(* CODESYS project filling_station_1808.ecp

Project tree, tasks and I/O mapping:
  GenericDummyMasterDevice : Generic Master, WAGO, order no. None, version 1.0.0.0
  PFC200_CS_2ETH_RS : 750-8202 PFC200 2ETH RS, WAGO, order no. 0750-8202, version 1.4.1.22
    application Application
      libraries: ; Util, * (System); VisuDialogs, * (System)
      task PLC_Task (cyclic, interval t#10ms, priority 14) calls PLC_PRG
      task Visu_Task (cyclic, interval t#10ms, priority 14) calls VISU_PRG
      function CONVERT_PRESSURE_TO_LEVEL [ST]
      visualisation Visualization
      function READ_PRESSURE [ST]
      global variables GVL
      function XOR_MANUAL_AUTOMATIC_VALVE_CONTROL [ST]
      function READ_VALVE_POSITION [ST]
      function AVOID_SIMULT_VALVE_OPEN_AND_CLOSE [ST]
      program PLC_PRG [FBD]
      image pool ImagePool
      visualisation Visualization_1
      function ASSIGN_OUTPUTS [ST]
      visualisation Visualization_2
      function ACTUATOR [ST]
    DeviceAdapter
    Kbus : Kbus, WAGO, version 1.3.0.0
        unmapped channels: K-BUS diagnostics
      _8_DO_Generic : 075x-8DO, WAGO, order no. 075x-8DO, version 0.0.0.11
          settings: K-BUS Module slot index = 1
          output vbOpenSamsonValve : BOOL  // _OUT._OUT
          output vbCloseSamsonValve : BOOL  // _OUT._OUT
          output vbOpenDrainValveAbovePump : BOOL  // _OUT._OUT
          output vbSwitchOnPump : BOOL  // _OUT._OUT
          unmapped channels: _OUT
        DeviceAdapter
      _4_AI_0_10V_DC_s_e : 0750-0459, WAGO, order no. 0750-0459, version 0.0.0.11
          settings: K-BUS Module slot index = 2
          input  vwRawValvePosition : WORD  // _IW 1
          unmapped channels: _IW 2, _IW 3, _IW 4
        DeviceAdapter
      _2_AI_4_20mA_Diff_Measurement_Input : 0750-0492, WAGO, order no. 0750-0492, version 0.0.0.7
          settings: K-BUS Module slot index = 3
          input  vwRawPressure : WORD  // _IW 1
          unmapped channels: _IW 2
        DeviceAdapter
    MODBUS
      MODBUS : MODBUS, WAGO, order no. n/a, version 1.1.1.13
    Serial
      COM1 : COM1, WAGO, version 0.0.0.19
  e_DISPLAY_7300T_WP_10_1_1280x800_PIO1 : 0762-3003 e!DISPLAY 7300T - WP 10.1, WAGO, order no. 0762-3003, version 0.0.0.3
    DeviceAdapter
  libraries: WagoVisuIcons, 1.0.0.7 (WAGO)
  text list GlobalTextList
  5ce3da45-db07-42e7-a21c-a00fff4ed8f6|C:\Users\Alexander Wilms\Documents\Ausbildung\Hochschule Darmstadt\Master Electrical Engineering\1. Semester\Team Project\team-project\40_Implementation\hydraulics-schematic-simplified.png
  5ce3da45-db07-42e7-a21c-a00fff4ed8f6|C:\Users\Alexander Wilms\Documents\Ausbildung\Hochschule Darmstadt\Master Electrical Engineering\1. Semester\Team Project\team-project\30_Architecture\hydraulics-schematic-simplified.png
*)

// PFC200_CS_2ETH_RS/Application/GVL
VAR_GLOBAL
	vrWaterLevel:REAL;
	vrgrWaterLevel:ARRAY[1..16] OF REAL;
	vrStandardGravity:REAL:=9.81;
	viDensityWater:INT:=1000;
	vrValvePosition:REAL;
	vrValvePositionPercentage:REAL;
	vrValvePositionDesired:REAL;
	viPumpPowerPercentage:INT;
	vbManualValveControl:BOOL:=TRUE;
	vbAutomaticValveControl:BOOL:=FALSE;
	vbPreviousValveControl:STRING:='MANUAL';
	vbPreviousSamsonValveDirection:STRING:='STOP';
	vbStopSamsonValve:BOOL:=TRUE;
	vbOpenSamsonValveCtrl:BOOL;
	vbCloseSamsonValveCtrl:BOOL;
	vbOpenDrainValveBelowVessel:BOOL:=FALSE;
	vbOpenDrainValveAbovePumpCtrl:BOOL:=FALSE;
	vbSwitchOnPumpCtrl:BOOL:=FALSE;
	vbTrash: BOOL;
	vrController_Level_SP:REAL;
	vrController_PV:REAL;
	vbController_Manual_Mode:BOOL:=FALSE;
	vrController_Output:REAL;
	vrController_Output_reversed:REAL;
	Water_Valve_Open: BOOL;
	Water_Valve_Close: BOOL;
	PID_1: PID;
END_VAR

// PFC200_CS_2ETH_RS/Application/PLC_PRG
PROGRAM PLC_PRG
VAR
	PID_0: PID;
	TRASH: BOOL;
END_VAR

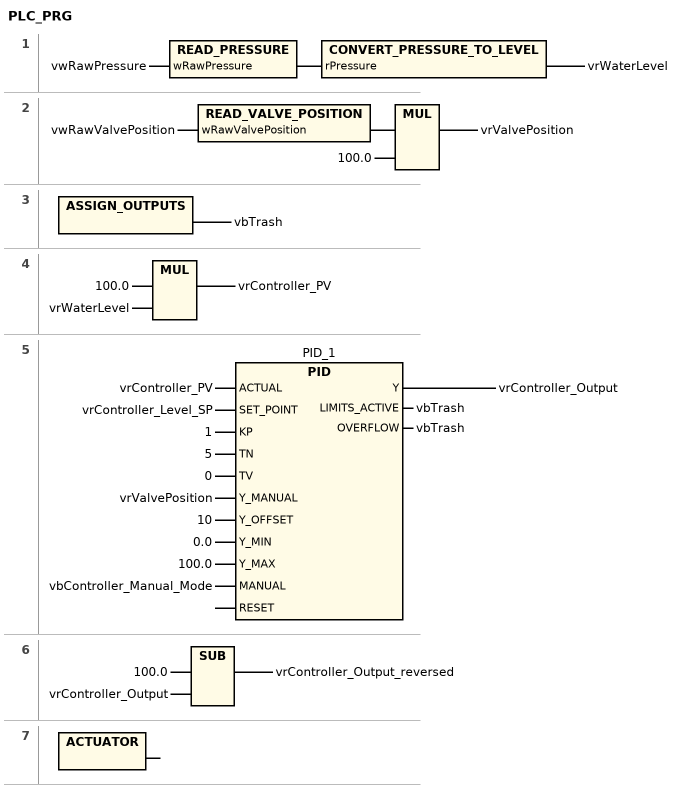
// NETWORK 1
vrWaterLevel := CONVERT_PRESSURE_TO_LEVEL(rPressure := READ_PRESSURE(wRawPressure := vwRawPressure));

// NETWORK 2
vrValvePosition := READ_VALVE_POSITION(wRawValvePosition := vwRawValvePosition) * 100.0;

// NETWORK 3
vbTrash := ASSIGN_OUTPUTS();

// NETWORK 4
vrController_PV := 100.0 * vrWaterLevel;

// NETWORK 5
PID_1(
    ACTUAL := vrController_PV,
    SET_POINT := vrController_Level_SP,
    KP := 1,
    TN := 5,
    TV := 0,
    Y_MANUAL := vrValvePosition,
    Y_OFFSET := 10,
    Y_MIN := 0.0,
    Y_MAX := 100.0,
    MANUAL := vbController_Manual_Mode,
    LIMITS_ACTIVE => vbTrash,
    OVERFLOW => vbTrash); // PID
vrController_Output := PID_1.Y;

// NETWORK 6
vrController_Output_reversed := 100.0 - vrController_Output;

// NETWORK 7
ACTUATOR();

END_PROGRAM

// PFC200_CS_2ETH_RS/Application/CONVERT_PRESSURE_TO_LEVEL
FUNCTION CONVERT_PRESSURE_TO_LEVEL : REAL
VAR_INPUT
	rPressure:REAL;
END_VAR
VAR
END_VAR

CONVERT_PRESSURE_TO_LEVEL := rPressure/viDensityWater/vrStandardGravity;

END_FUNCTION

// PFC200_CS_2ETH_RS/Application/READ_PRESSURE
FUNCTION READ_PRESSURE : REAL
VAR_INPUT
	wRawPressure:WORD;
END_VAR
VAR
END_VAR

READ_PRESSURE := WORD_TO_REAL((wRawPressure)*9800)/65535;

END_FUNCTION

// PFC200_CS_2ETH_RS/Application/READ_VALVE_POSITION
FUNCTION READ_VALVE_POSITION : REAL
VAR_INPUT
	wRawValvePosition:WORD;
END_VAR
VAR
END_VAR

READ_VALVE_POSITION := WORD_TO_REAL(wRawValvePosition)/65535;
vrValvePositionPercentage := READ_VALVE_POSITION*100;

END_FUNCTION

// PFC200_CS_2ETH_RS/Application/ASSIGN_OUTPUTS
FUNCTION ASSIGN_OUTPUTS : BOOL
VAR_INPUT
END_VAR
VAR
END_VAR

vbSwitchOnPump:=vbSwitchOnPumpCtrl;
vbOpenDrainValveAbovePump:=vbOpenDrainValveAbovePumpCtrl;
vbOpenSamsonValveCtrl:=vbOpenSamsonValve;
vbCloseSamsonValveCtrl:=vbCloseSamsonValve;
ASSIGN_OUTPUTS:=TRUE;

END_FUNCTION

// PFC200_CS_2ETH_RS/Application/ACTUATOR
FUNCTION ACTUATOR : BOOL
VAR_INPUT
END_VAR
VAR
END_VAR

IF (vrController_Output_reversed - vrValvePosition) <= 2 AND (  vrValvePosition - vrController_Output_reversed ) <=2
THEN
vbOpenSamsonValve:=vbOpenSamsonValve;
vbCloseSamsonValve:=vbCloseSamsonValve;
ELSIF
(vrController_Output_reversed - vrValvePosition) >2
THEN
vbOpenSamsonValve:=TRUE;
vbCloseSamsonValve:=FALSE;
ELSE
vbOpenSamsonValve:=FALSE;
vbCloseSamsonValve:=TRUE;
END_IF

END_FUNCTION

// PFC200_CS_2ETH_RS/Application/XOR_MANUAL_AUTOMATIC_VALVE_CONTROL
FUNCTION XOR_MANUAL_AUTOMATIC_VALVE_CONTROL : BOOL
VAR_INPUT
END_VAR
VAR
END_VAR

IF vbAutomaticValveControl AND vbManualValveControl THEN
	IF vbPreviousValveControl = 'MANUAL' THEN
			vbAutomaticValveControl := TRUE;
			vbManualValveControl := FALSE;
			vbPreviousValveControl := 'AUTOMATIC';
	ELSIF
			vbPreviousValveControl =  'AUTOMATIC' THEN
			vbAutomaticValveControl := FALSE;
			vbManualValveControl := TRUE;
			vbPreviousValveControl := 'MANUAL';
	END_IF
END_IF

XOR_MANUAL_AUTOMATIC_VALVE_CONTROL := TRUE;

END_FUNCTION

// PFC200_CS_2ETH_RS/Application/AVOID_SIMULT_VALVE_OPEN_AND_CLOSE
FUNCTION AVOID_SIMULT_VALVE_OPEN_AND_CLOSE : BOOL
VAR_INPUT
END_VAR
VAR
END_VAR

IF vbOpenSamsonValve AND vbStopSamsonValve THEN
	IF vbPreviousSamsonValveDirection = 'OPEN' THEN
		vbOpenSamsonValve := FALSE;
		vbStopSamsonValve := TRUE;
		vbCloseSamsonValve := FALSE;
		vbPreviousSamsonValveDirection := 'STOP';
	ELSIF vbPreviousSamsonValveDirection = 'STOP' THEN
		vbOpenSamsonValve := TRUE;
		vbStopSamsonValve := FALSE;
		vbCloseSamsonValve := FALSE;
		vbPreviousSamsonValveDirection := 'OPEN';
	END_IF
ELSIF vbStopSamsonValve AND vbCloseSamsonValve THEN
	IF vbPreviousSamsonValveDirection = 'STOP' THEN
		vbOpenSamsonValve := FALSE;
		vbStopSamsonValve := FALSE;
		vbCloseSamsonValve := TRUE;
		vbPreviousSamsonValveDirection := 'CLOSE';
	ELSIF vbPreviousSamsonValveDirection = 'CLOSE' THEN
		vbOpenSamsonValve := FALSE;
		vbStopSamsonValve := TRUE;
		vbCloseSamsonValve := FALSE;
		vbPreviousSamsonValveDirection := 'STOP';
	END_IF
ELSIF vbOpenSamsonValve AND vbCloseSamsonValve THEN
	IF vbPreviousSamsonValveDirection = 'OPEN' THEN
		vbOpenSamsonValve := FALSE;
		vbStopSamsonValve := FALSE;
		vbCloseSamsonValve := TRUE;
		vbPreviousSamsonValveDirection := 'CLOSE';
	ELSIF vbPreviousSamsonValveDirection = 'CLOSE' THEN
		vbOpenSamsonValve := TRUE;
		vbStopSamsonValve := FALSE;
		vbCloseSamsonValve := FALSE;
		vbPreviousSamsonValveDirection := 'OPEN';
	END_IF
END_IF

AVOID_SIMULT_VALVE_OPEN_AND_CLOSE := TRUE;

END_FUNCTION

// PFC200_CS_2ETH_RS/Application/Visualization
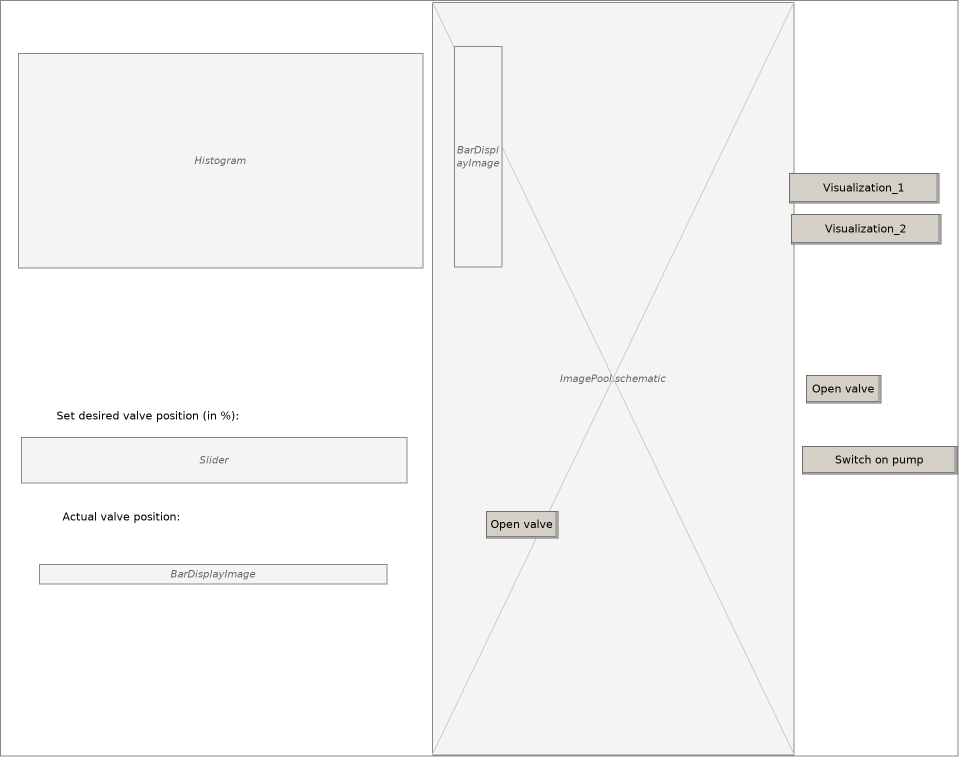
VISUALIZATION Visualization  // 959x757
    Image (432,2 362x753), image: ImagePool.schematic
    BarDisplayImage (454,46 48x221), value: vrWaterLevel, style: BarDisplayImage-Gray, scale format: %.1f, scale 0..1
        p518627256: m
    Histogram (18,53 405x215), scale format: %.1f, scale 0..1
        p1518820177: vrgrWaterLevel
        p102497268: vrgrWaterLevel
        p788070771: ARRAY [1..16] OF REAL
    Button (806,375 75x28), "Open valve"
        toggle vbOpenDrainValveAbovePumpCtrl
    Button (802,446 155x28), "Switch on pump"
        toggle vbSwitchOnPumpCtrl
    Label (61,407 174x18), "Set desired valve position (in %):"
    Slider (21,437 386x46), variable: vrValvePositionDesired, scale 0..100
    Button (486,511 72x27), "Open valve"
        toggle vbOpenDrainValveBelowVessel
    BarDisplayImage (39,564 348x20), value: vrWaterLevel, style: BarDisplayImage-Gray, scale format: %i, scale 0..100
        p518627256: m
    Label (59,508 125x18), "Actual valve position:"
    Button (789,173 150x30), "Visualization_1"
        OnMouseClick:  Assign=Visualization_1, Type=Assignment
    Button (791,214 150x30), "Visualization_2"
        OnMouseClick:  Assign=Visualization_2, Type=Assignment
END_VISUALIZATION

// PFC200_CS_2ETH_RS/Application/Visualization_1
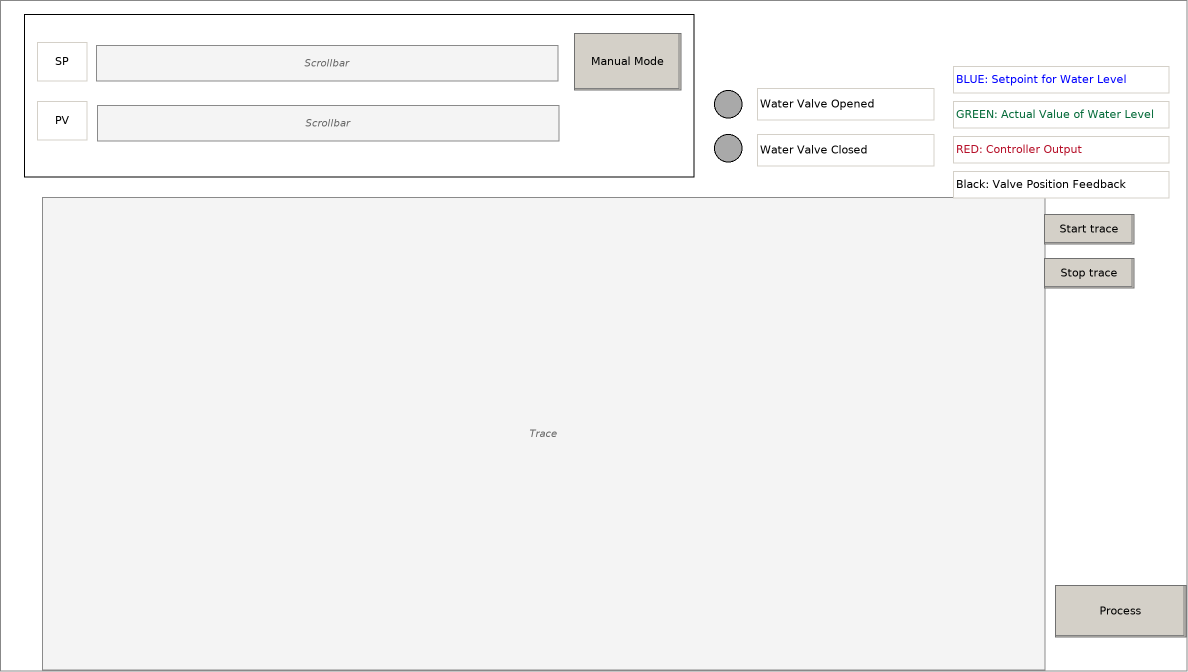
VISUALIZATION Visualization_1  // 1188x672
VAR_IN_OUT
END_VAR
VAR
	bResetTrigger : BOOL;
	bStart : BOOL;
	bStop : BOOL;
	bStore : BOOL;
	sStoreFilename : STRING;
	bRestore : BOOL;
	sRestoreFilename : STRING;
END_VAR
    RoundedRectangle (24,14 670x163)
    Button (1055,585 131x52), "Process"
        OnMouseClick:  Assign=Visualization, Type=Assignment
    Scrollbar (96,45 462x36), text variable: vrController_Level_SP
        p1057716461: vrController_Level_SP
        p2175578022: vrController_Level_SP
    Trace (42,197 1003x473)
        p3825648158: bResetTrigger
        p866368322: bStart
        p3851742229: bStop
        p2132035699: bStore
        p163910951: sStoreFilename
        p2217859334: bRestore
        p1301606187: sRestoreFilename
    Button (1044,214 90x30), "Start trace"
        toggle bStart
    Button (1044,258 90x30), "Stop trace"
        toggle bStop
    Textfield (953,66 216x27), "BLUE: Setpoint for Water Level"
    Textfield (953,101 216x27), "GREEN: Actual Value of Water Level"
    Textfield (953,136 216x27), "RED: Controller Output"
    Textfield (953,171 216x27), "Black: Valve Position Feedback"
    Button (574,33 107x57), "Manual Mode", colour toggle: vbController_Manual_Mode
        OnMouseClick:  ToggleVariable=vbController_Manual_Mode
        OnDialogClosed:  ToggleVariable=vbController_Manual_Mode
    Ellipse (714,90 28x28), colour toggle: vbOpenSamsonValveCtrl
    Ellipse (714,134 28x28), colour toggle: vbCloseSamsonValveCtrl
    Textfield (757,88 177x32), "Water Valve Opened"
    Textfield (757,134 177x32), "Water Valve Closed"
    Textfield (37,42 50x39), "SP"
    Textfield (37,101 50x39), "PV"
    Scrollbar (97,105 462x36), text variable: vrController_Level_SP
        p1057716461: vrController_PV
        p2175578022: vrController_Level_SP
END_VISUALIZATION

// PFC200_CS_2ETH_RS/Application/Visualization_2
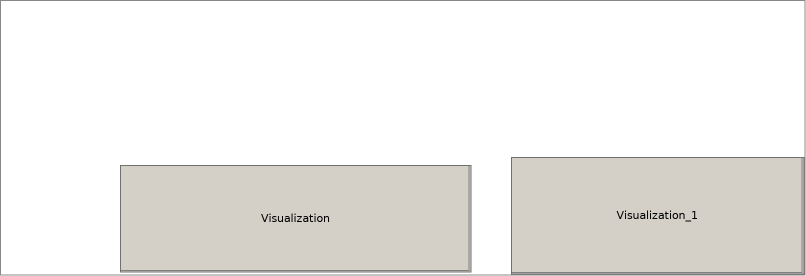
VISUALIZATION Visualization_2  // 806x276
    Button (120,165 351x107), "Visualization"
        OnMouseClick:  Assign=Visualization, Type=Assignment
    Button (511,157 293x117), "Visualization_1"
        OnMouseClick:  Assign=Visualization_1, Type=Assignment
END_VISUALIZATION
